// LS Electric XG5000 project: MODBUS_PR_3차프로젝트 최종최종
// PLC LSPLC
// module base 0 slot 0: 입출력 모듈:XBC-DR32H (DC 24V 입력, 릴레이 출력 32점)

PROGRAM 구동부_사본 (task: 스캔 프로그램)

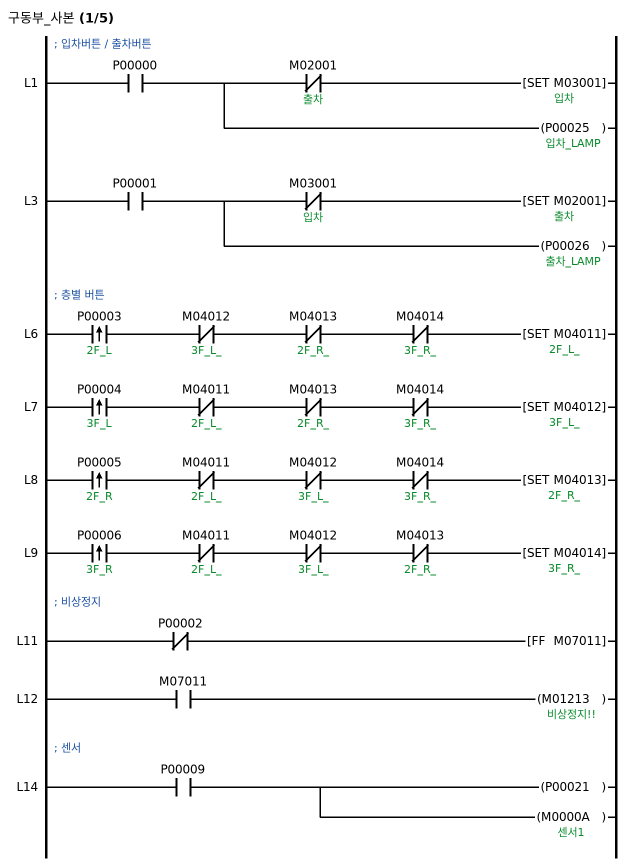
// 입차버튼 / 출차버튼
; L1
LOAD      P00000
MPUSH
AND NOT   M02001	// 출차
SET       M03001	// 입차
MPOP
OUT       P00025	// 입차_LAMP
; L3
LOAD      P00001
MPUSH
AND NOT   M03001	// 입차
SET       M02001	// 출차
MPOP
OUT       P00026	// 출차_LAMP
// 층별 버튼
; L6
LOADP     P00003	// 2F_L
AND NOT   M04012	// 3F_L_
AND NOT   M04013	// 2F_R_
AND NOT   M04014	// 3F_R_
SET       M04011	// 2F_L_
; L7
LOADP     P00004	// 3F_L
AND NOT   M04011	// 2F_L_
AND NOT   M04013	// 2F_R_
AND NOT   M04014	// 3F_R_
SET       M04012	// 3F_L_
; L8
LOADP     P00005	// 2F_R
AND NOT   M04011	// 2F_L_
AND NOT   M04012	// 3F_L_
AND NOT   M04014	// 3F_R_
SET       M04013	// 2F_R_
; L9
LOADP     P00006	// 3F_R
AND NOT   M04011	// 2F_L_
AND NOT   M04012	// 3F_L_
AND NOT   M04013	// 2F_R_
SET       M04014	// 3F_R_
// 비상정지
; L11
LOAD NOT  P00002
FF        M07011
; L12
LOAD      M07011
OUT       M01213	// 비상정지!!
// 센서
; L14
LOAD      P00009
OUT       P00021
OUT       M0000A	// 센서1

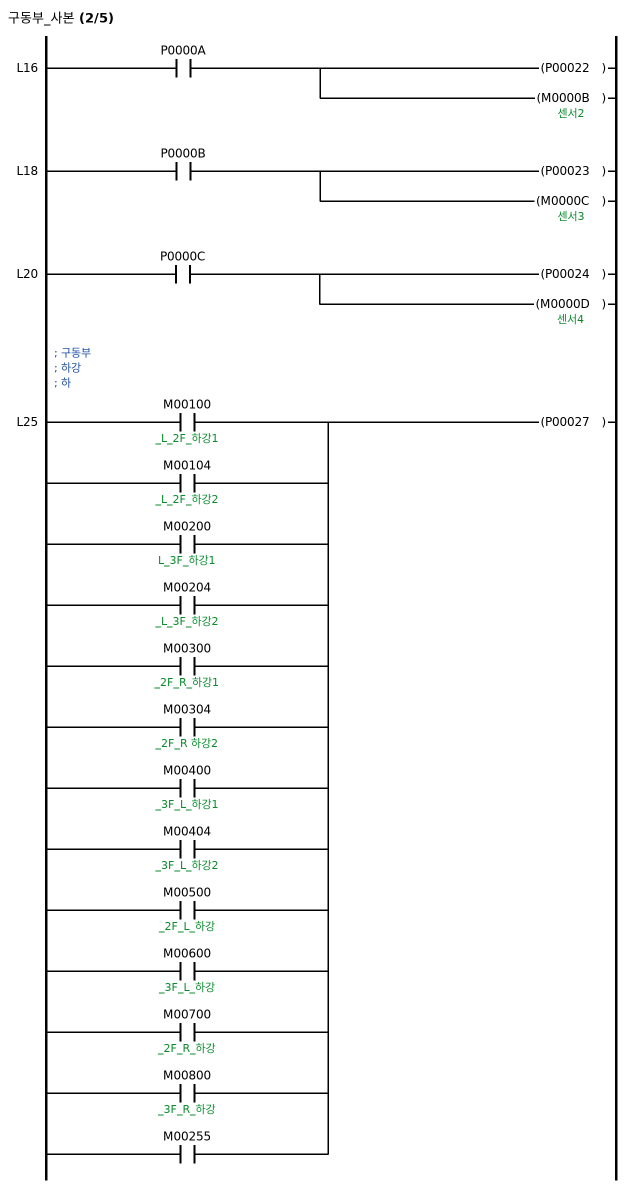
; L16
LOAD      P0000A
OUT       P00022
OUT       M0000B	// 센서2
; L18
LOAD      P0000B
OUT       P00023
OUT       M0000C	// 센서3
; L20
LOAD      P0000C
OUT       P00024
OUT       M0000D	// 센서4
// 구동부
// 하강
; L25
LOAD      M00100	// _L_2F_하강1
OR        M00104	// _L_2F_하강2
OR        M00200	// L_3F_하강1
OR        M00204	// _L_3F_하강2
OR        M00300	// _2F_R_하강1
OR        M00304	// _2F_R 하강2
OR        M00400	// _3F_L_하강1
OR        M00404	// _3F_L_하강2
OR        M00500	// _2F_L_하강
OR        M00600	// _3F_L_하강
OR        M00700	// _2F_R_하강
OR        M00800	// _3F_R_하강
OR        M00255
OUT       P00027
// output comment: 하

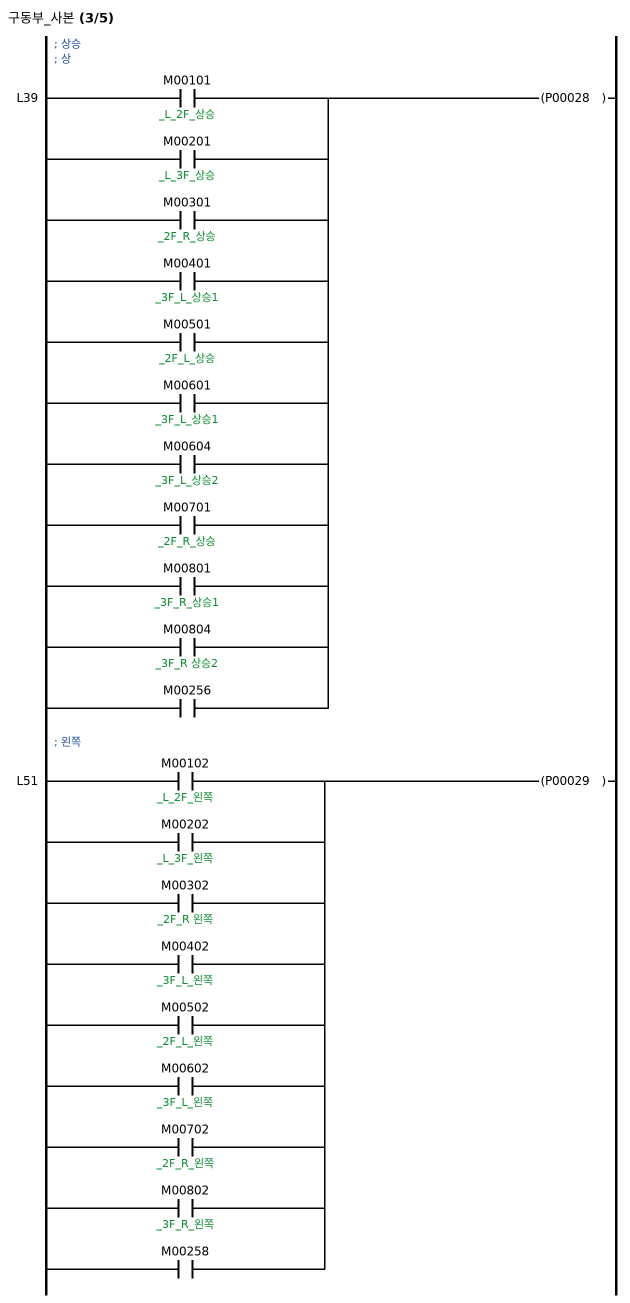
// 상승
; L39
LOAD      M00101	// _L_2F_상승
OR        M00201	// _L_3F_상승
OR        M00301	// _2F_R_상승
OR        M00401	// _3F_L_상승1
OR        M00501	// _2F_L_상승
OR        M00601	// _3F_L_상승1
OR        M00604	// _3F_L_상승2
OR        M00701	// _2F_R_상승
OR        M00801	// _3F_R_상승1
OR        M00804	// _3F_R 상승2
OR        M00256
OUT       P00028
// output comment: 상
// 왼쪽
; L51
LOAD      M00102	// _L_2F_왼쪽
OR        M00202	// _L_3F_왼쪽
OR        M00302	// _2F_R 왼쪽
OR        M00402	// _3F_L_왼쪽
OR        M00502	// _2F_L_왼쪽
OR        M00602	// _3F_L_왼쪽
OR        M00702	// _2F_R_왼쪽
OR        M00802	// _3F_R_왼쪽
OR        M00258
OUT       P00029

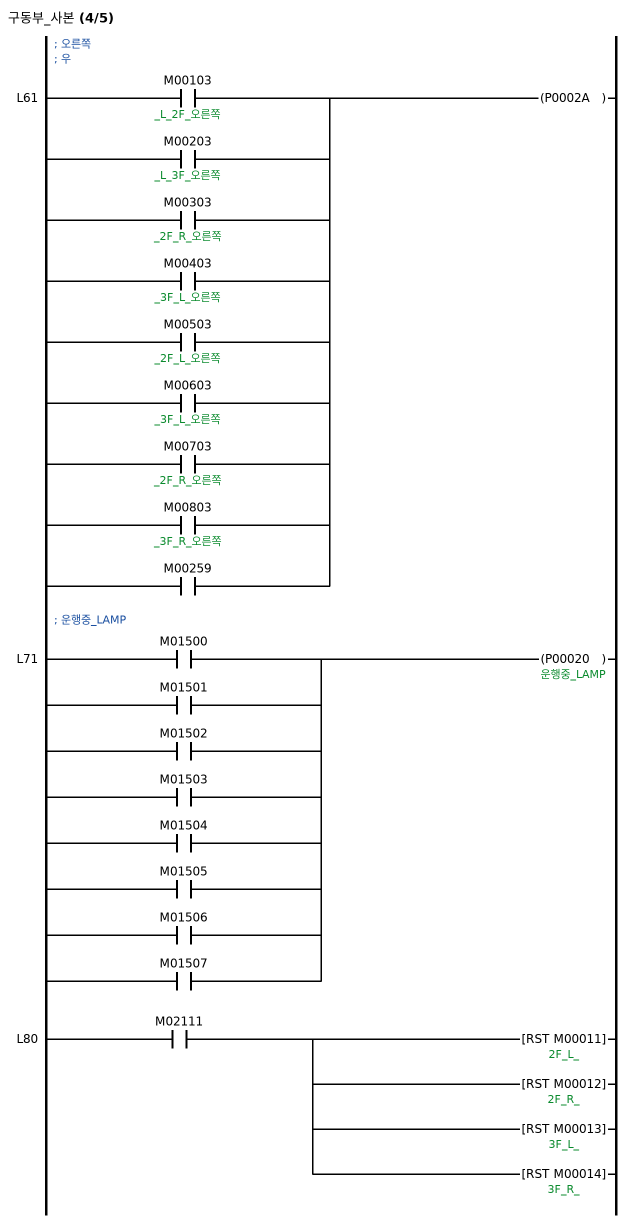
// 오른쪽
; L61
LOAD      M00103	// _L_2F_오른쪽
OR        M00203	// _L_3F_오른쪽
OR        M00303	// _2F_R_오른쪽
OR        M00403	// _3F_L_오른쪽
OR        M00503	// _2F_L_오른쪽
OR        M00603	// _3F_L_오른쪽
OR        M00703	// _2F_R_오른쪽
OR        M00803	// _3F_R_오른쪽
OR        M00259
OUT       P0002A
// output comment: 우
// 운행중_LAMP
; L71
LOAD      M01500
OR        M01501
OR        M01502
OR        M01503
OR        M01504
OR        M01505
OR        M01506
OR        M01507
OUT       P00020	// 운행중_LAMP
; L80
LOAD      M02111
RST       M00011	// 2F_L_
RST       M00012	// 2F_R_
RST       M00013	// 3F_L_
RST       M00014	// 3F_R_

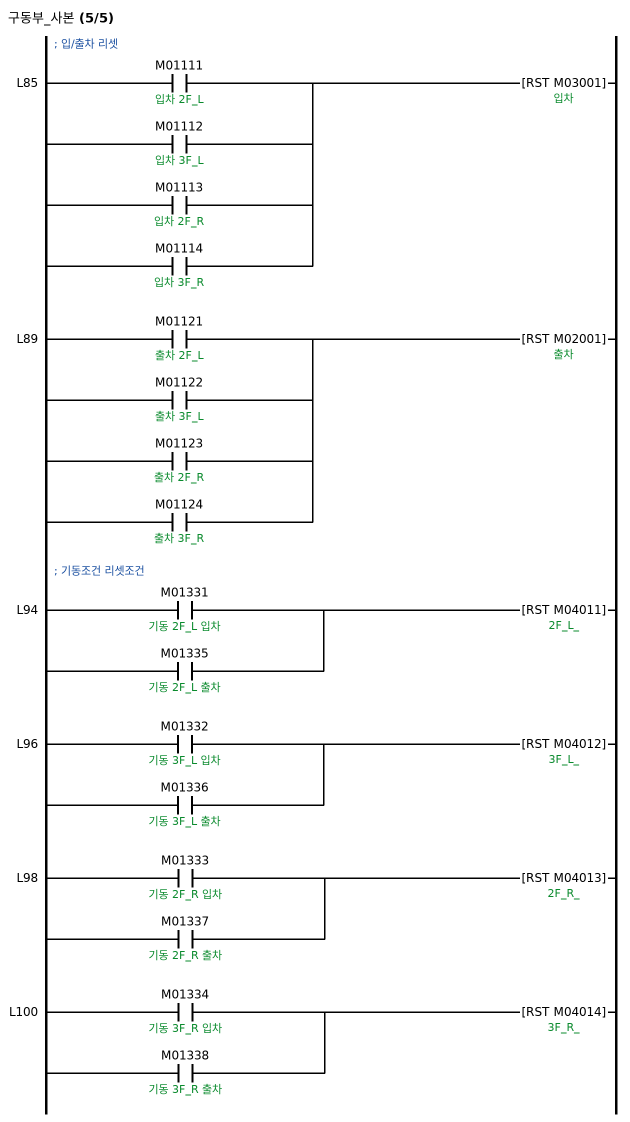
// 입/출차 리셋
; L85
LOAD      M01111	// 입차 2F_L 
OR        M01112	// 입차 3F_L
OR        M01113	// 입차 2F_R
OR        M01114	// 입차 3F_R
RST       M03001	// 입차
; L89
LOAD      M01121	// 출차 2F_L
OR        M01122	// 출차 3F_L
OR        M01123	// 출차 2F_R
OR        M01124	// 출차 3F_R
RST       M02001	// 출차
// 기동조건 리셋조건
; L94
LOAD      M01331	// 기동 2F_L 입차
OR        M01335	// 기동 2F_L 출차
RST       M04011	// 2F_L_
; L96
LOAD      M01332	// 기동 3F_L 입차
OR        M01336	// 기동 3F_L 출차
RST       M04012	// 3F_L_
; L98
LOAD      M01333	// 기동 2F_R 입차
OR        M01337	// 기동 2F_R 출차
RST       M04013	// 2F_R_
; L100
LOAD      M01334	// 기동 3F_R 입차
OR        M01338	// 기동 3F_R 출차
RST       M04014	// 3F_R_

PROGRAM 출차 (task: 스캔 프로그램)

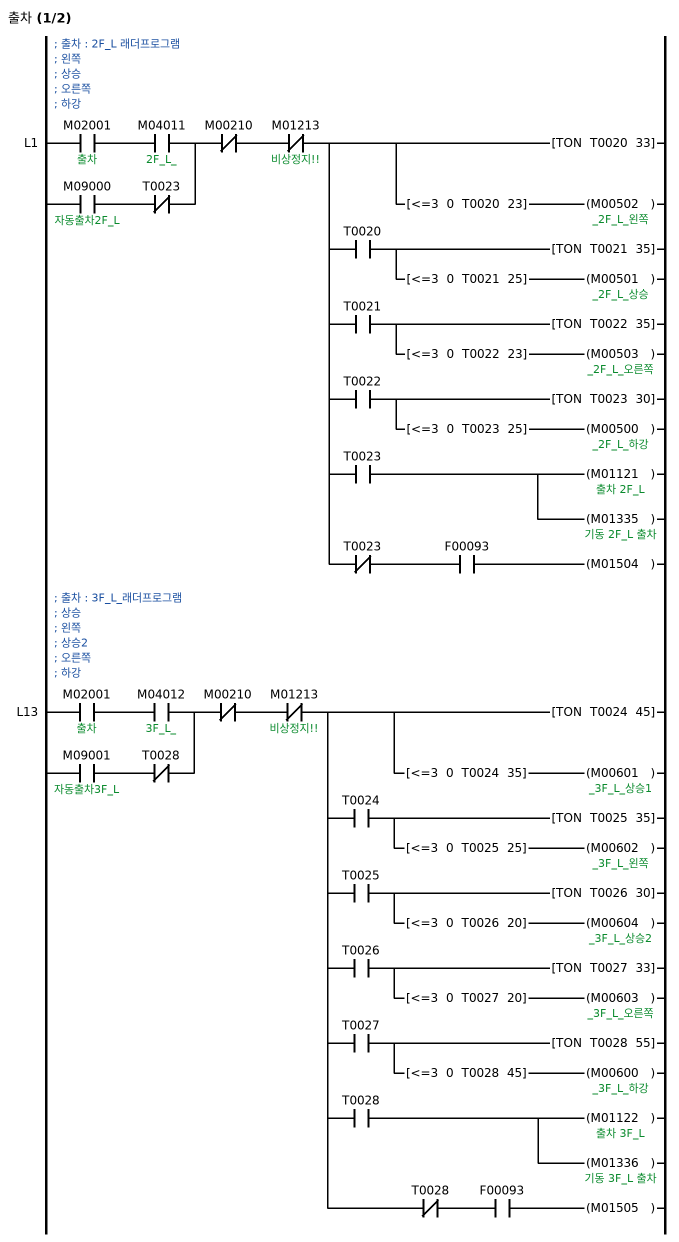
// 출차 : 2F_L 래더프로그램
; L1
LOAD      M02001	// 출차
AND       M04011	// 2F_L_
LOAD      M09000	// 자동출차2F_L
AND NOT   T0023
OR LOAD
AND NOT   M00210
AND NOT   M01213	// 비상정지!!
TON       T0020 33
MPUSH
AND<=3    0 T0020 23
OUT       M00502	// _2F_L_왼쪽
MLOAD
AND       T0020
TON       T0021 35
AND<=3    0 T0021 25
OUT       M00501	// _2F_L_상승
MLOAD
AND       T0021
TON       T0022 35
AND<=3    0 T0022 23
OUT       M00503	// _2F_L_오른쪽
MLOAD
AND       T0022
TON       T0023 30
AND<=3    0 T0023 25
OUT       M00500	// _2F_L_하강
MLOAD
AND       T0023
OUT       M01121	// 출차 2F_L
OUT       M01335	// 기동 2F_L 출차
MPOP
AND NOT   T0023
AND       F00093
OUT       M01504
// output comment: 왼쪽
// output comment: 상승
// output comment: 오른쪽
// output comment: 하강
// 출차 : 3F_L_래더프로그램
; L13
LOAD      M02001	// 출차
AND       M04012	// 3F_L_
LOAD      M09001	// 자동출차3F_L
AND NOT   T0028
OR LOAD
AND NOT   M00210
AND NOT   M01213	// 비상정지!!
TON       T0024 45
MPUSH
AND<=3    0 T0024 35
OUT       M00601	// _3F_L_상승1
MLOAD
AND       T0024
TON       T0025 35
AND<=3    0 T0025 25
OUT       M00602	// _3F_L_왼쪽
MLOAD
AND       T0025
TON       T0026 30
AND<=3    0 T0026 20
OUT       M00604	// _3F_L_상승2
MLOAD
AND       T0026
TON       T0027 33
AND<=3    0 T0027 20
OUT       M00603	// _3F_L_오른쪽
MLOAD
AND       T0027
TON       T0028 55
AND<=3    0 T0028 45
OUT       M00600	// _3F_L_하강
MLOAD
AND       T0028
OUT       M01122	// 출차 3F_L
OUT       M01336	// 기동 3F_L 출차
MPOP
AND NOT   T0028
AND       F00093
OUT       M01505
// output comment: 상승
// output comment: 왼쪽
// output comment: 상승2
// output comment: 오른쪽
// output comment: 하강

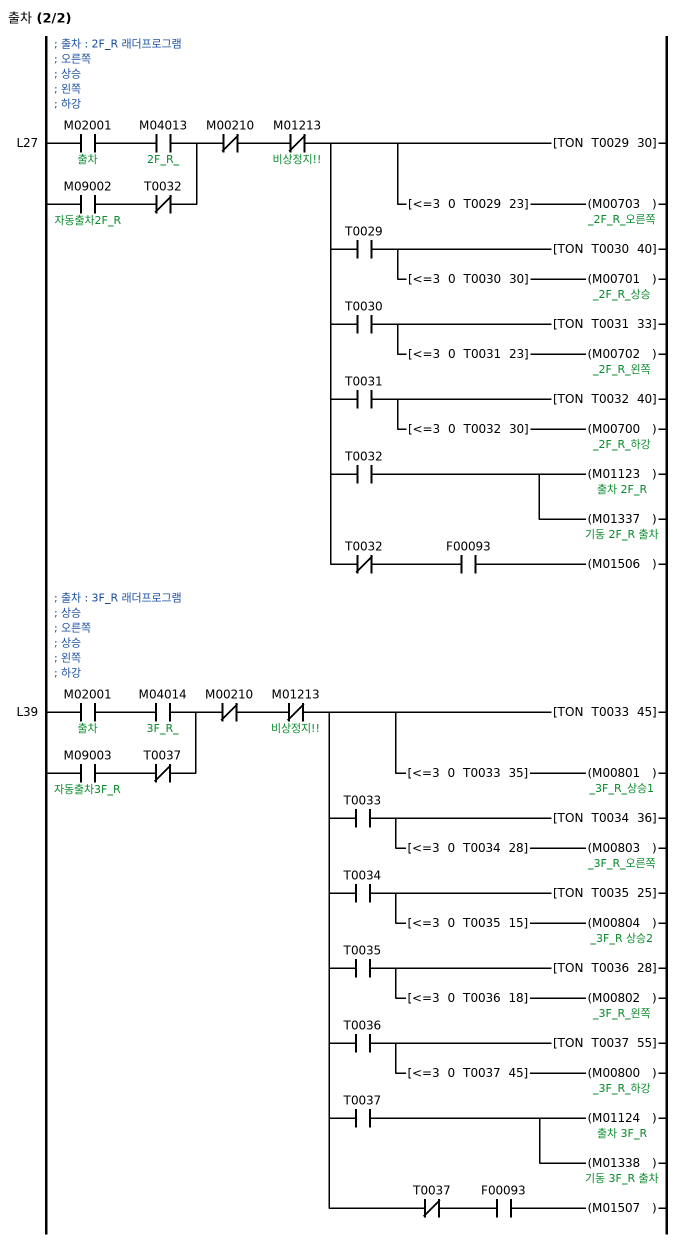
// 출차 : 2F_R 래더프로그램
; L27
LOAD      M02001	// 출차
AND       M04013	// 2F_R_
LOAD      M09002	// 자동출차2F_R
AND NOT   T0032
OR LOAD
AND NOT   M00210
AND NOT   M01213	// 비상정지!!
TON       T0029 30
MPUSH
AND<=3    0 T0029 23
OUT       M00703	// _2F_R_오른쪽
MLOAD
AND       T0029
TON       T0030 40
AND<=3    0 T0030 30
OUT       M00701	// _2F_R_상승
MLOAD
AND       T0030
TON       T0031 33
AND<=3    0 T0031 23
OUT       M00702	// _2F_R_왼쪽
MLOAD
AND       T0031
TON       T0032 40
AND<=3    0 T0032 30
OUT       M00700	// _2F_R_하강
MLOAD
AND       T0032
OUT       M01123	// 출차 2F_R
OUT       M01337	// 기동 2F_R 출차
MPOP
AND NOT   T0032
AND       F00093
OUT       M01506
// output comment: 오른쪽
// output comment: 상승
// output comment: 왼쪽
// output comment: 하강
// 출차 : 3F_R 래더프로그램
; L39
LOAD      M02001	// 출차
AND       M04014	// 3F_R_
LOAD      M09003	// 자동출차3F_R
AND NOT   T0037
OR LOAD
AND NOT   M00210
AND NOT   M01213	// 비상정지!!
TON       T0033 45
MPUSH
AND<=3    0 T0033 35
OUT       M00801	// _3F_R_상승1
MLOAD
AND       T0033
TON       T0034 36
AND<=3    0 T0034 28
OUT       M00803	// _3F_R_오른쪽
MLOAD
AND       T0034
TON       T0035 25
AND<=3    0 T0035 15
OUT       M00804	// _3F_R 상승2
MLOAD
AND       T0035
TON       T0036 28
AND<=3    0 T0036 18
OUT       M00802	// _3F_R_왼쪽
MLOAD
AND       T0036
TON       T0037 55
AND<=3    0 T0037 45
OUT       M00800	// _3F_R_하강
MLOAD
AND       T0037
OUT       M01124	// 출차 3F_R
OUT       M01338	// 기동 3F_R 출차
MPOP
AND NOT   T0037
AND       F00093
OUT       M01507
// output comment: 상승
// output comment: 오른쪽
// output comment: 상승
// output comment: 왼쪽
// output comment: 하강

PROGRAM 입차 (task: 스캔 프로그램)

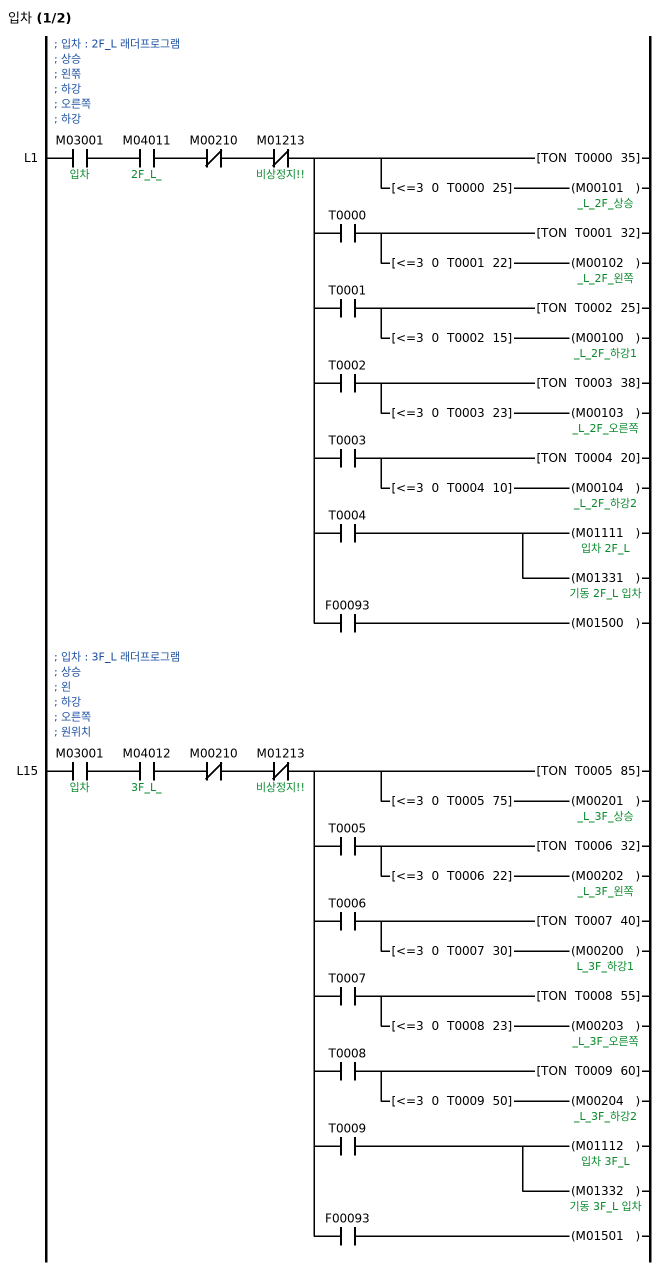
// 입차 : 2F_L 래더프로그램
; L1
LOAD      M03001	// 입차
AND       M04011	// 2F_L_
AND NOT   M00210
AND NOT   M01213	// 비상정지!!
TON       T0000 35
MPUSH
AND<=3    0 T0000 25
OUT       M00101	// _L_2F_상승
MLOAD
AND       T0000
TON       T0001 32
AND<=3    0 T0001 22
OUT       M00102	// _L_2F_왼쪽
MLOAD
AND       T0001
TON       T0002 25
AND<=3    0 T0002 15
OUT       M00100	// _L_2F_하강1
MLOAD
AND       T0002
TON       T0003 38
AND<=3    0 T0003 23
OUT       M00103	// _L_2F_오른쪽
MLOAD
AND       T0003
TON       T0004 20
AND<=3    0 T0004 10
OUT       M00104	// _L_2F_하강2
MLOAD
AND       T0004
OUT       M01111	// 입차 2F_L 
OUT       M01331	// 기동 2F_L 입차
MPOP
AND       F00093
OUT       M01500
// output comment: 상승
// output comment: 왼쪾
// output comment: 하강
// output comment: 오른쪽
// output comment: 하강
// 입차 : 3F_L 래더프로그램
; L15
LOAD      M03001	// 입차
AND       M04012	// 3F_L_
AND NOT   M00210
AND NOT   M01213	// 비상정지!!
TON       T0005 85
MPUSH
AND<=3    0 T0005 75
OUT       M00201	// _L_3F_상승
MLOAD
AND       T0005
TON       T0006 32
AND<=3    0 T0006 22
OUT       M00202	// _L_3F_왼쪽
MLOAD
AND       T0006
TON       T0007 40
AND<=3    0 T0007 30
OUT       M00200	// L_3F_하강1
MLOAD
AND       T0007
TON       T0008 55
AND<=3    0 T0008 23
OUT       M00203	// _L_3F_오른쪽
MLOAD
AND       T0008
TON       T0009 60
AND<=3    0 T0009 50
OUT       M00204	// _L_3F_하강2
MLOAD
AND       T0009
OUT       M01112	// 입차 3F_L
OUT       M01332	// 기동 3F_L 입차
MPOP
AND       F00093
OUT       M01501
// output comment: 상승
// output comment: 왼
// output comment: 하강
// output comment: 오른쪽
// output comment: 원위치

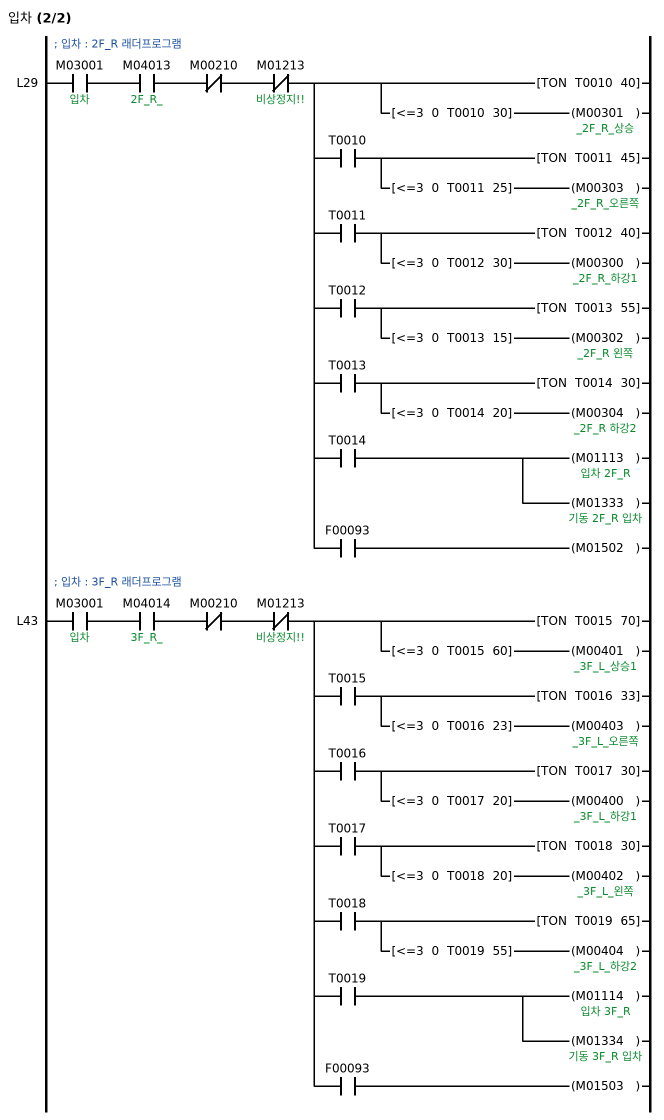
// 입차 : 2F_R 래더프로그램
; L29
LOAD      M03001	// 입차
AND       M04013	// 2F_R_
AND NOT   M00210
AND NOT   M01213	// 비상정지!!
TON       T0010 40
MPUSH
AND<=3    0 T0010 30
OUT       M00301	// _2F_R_상승
MLOAD
AND       T0010
TON       T0011 45
AND<=3    0 T0011 25
OUT       M00303	// _2F_R_오른쪽
MLOAD
AND       T0011
TON       T0012 40
AND<=3    0 T0012 30
OUT       M00300	// _2F_R_하강1
MLOAD
AND       T0012
TON       T0013 55
AND<=3    0 T0013 15
OUT       M00302	// _2F_R 왼쪽
MLOAD
AND       T0013
TON       T0014 30
AND<=3    0 T0014 20
OUT       M00304	// _2F_R 하강2
MLOAD
AND       T0014
OUT       M01113	// 입차 2F_R
OUT       M01333	// 기동 2F_R 입차
MPOP
AND       F00093
OUT       M01502
// 입차 : 3F_R 래더프로그램
; L43
LOAD      M03001	// 입차
AND       M04014	// 3F_R_
AND NOT   M00210
AND NOT   M01213	// 비상정지!!
TON       T0015 70
MPUSH
AND<=3    0 T0015 60
OUT       M00401	// _3F_L_상승1
MLOAD
AND       T0015
TON       T0016 33
AND<=3    0 T0016 23
OUT       M00403	// _3F_L_오른쪽
MLOAD
AND       T0016
TON       T0017 30
AND<=3    0 T0017 20
OUT       M00400	// _3F_L_하강1
MLOAD
AND       T0017
TON       T0018 30
AND<=3    0 T0018 20
OUT       M00402	// _3F_L_왼쪽
MLOAD
AND       T0018
TON       T0019 65
AND<=3    0 T0019 55
OUT       M00404	// _3F_L_하강2
MLOAD
AND       T0019
OUT       M01114	// 입차 3F_R
OUT       M01334	// 기동 3F_R 입차
MPOP
AND       F00093
OUT       M01503

PROGRAM 00.Initialize (task: 스캔 프로그램)

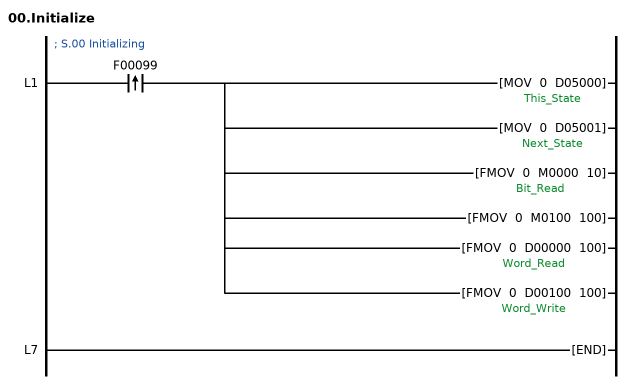
// S.00 Initializing
; L1
LOADP     F00099
MOV       0 D05000	// This_State
MOV       0 D05001	// Next_State
FMOV      0 M0000 10	// Bit_Read
FMOV      0 M0100 100
FMOV      0 D00000 100	// Word_Read
FMOV      0 D00100 100	// Word_Write
; L7
END

PROGRAM 10.Main (task: 스캔 프로그램)

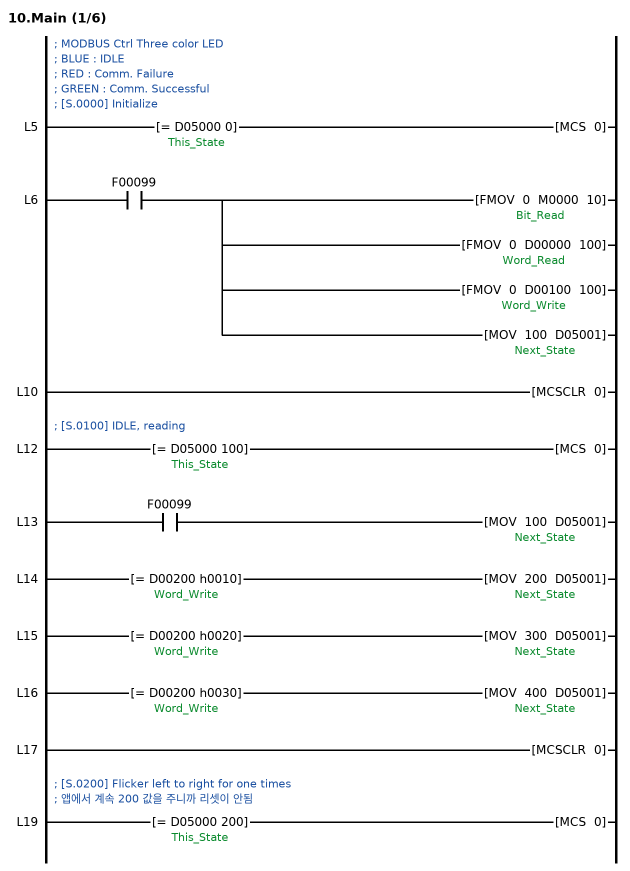
// MODBUS Ctrl Three color LED
// BLUE : IDLE
// RED : Comm. Failure
// GREEN : Comm. Successful
// [S.0000] Initialize
; L5
LOAD=     D05000 0	// This_State
MCS       0
; L6
LOAD      F00099
FMOV      0 M0000 10	// Bit_Read
FMOV      0 D00000 100	// Word_Read
FMOV      0 D00100 100	// Word_Write
MOV       100 D05001	// Next_State
; L10
MCSCLR    0
// [S.0100] IDLE, reading
; L12
LOAD=     D05000 100	// This_State
MCS       0
; L13
LOAD      F00099
MOV       100 D05001	// Next_State
; L14
LOAD=     D00200 h0010	// Word_Write
MOV       200 D05001	// Next_State
; L15
LOAD=     D00200 h0020	// Word_Write
MOV       300 D05001	// Next_State
; L16
LOAD=     D00200 h0030	// Word_Write
MOV       400 D05001	// Next_State
; L17
MCSCLR    0
// [S.0200] Flicker left to right for one times
; L19
LOAD=     D05000 200	// This_State
MCS       0
// output comment: 앱에서 계속 200 값을 주니까 리셋이 안됨

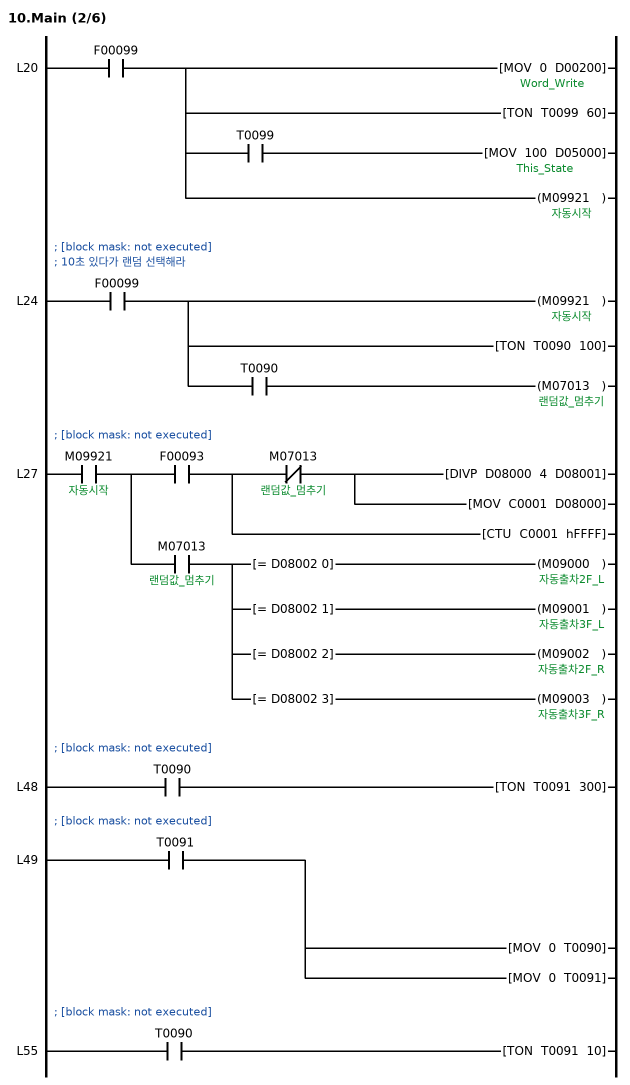
; L20
LOAD      F00099
MOV       0 D00200	// Word_Write
TON       T0099 60
MPUSH
AND       T0099
MOV       100 D05000	// This_State
MPOP
OUT       M09921	// 자동시작
; L24 (block mask: not executed)
LOAD      F00099
OUT       M09921	// 자동시작
TON       T0090 100
AND       T0090
OUT       M07013	// 랜덤값_멈추기
// output comment: 10초 있다가 랜덤 선택해라
; L27 (block mask: not executed)
LOAD      M09921	// 자동시작
MPUSH
AND       F00093
MPUSH
AND NOT   M07013	// 랜덤값_멈추기
DIVP      D08000 4 D08001
MOV       C0001 D08000
MPOP
CTU       C0001 hFFFF
MPOP
AND       M07013	// 랜덤값_멈추기
MPUSH
AND=      D08002 0
OUT       M09000	// 자동출차2F_L
MLOAD
AND=      D08002 1
OUT       M09001	// 자동출차3F_L
MLOAD
AND=      D08002 2
OUT       M09002	// 자동출차2F_R
MPOP
AND=      D08002 3
OUT       M09003	// 자동출차3F_R
; L48 (block mask: not executed)
LOAD      T0090
TON       T0091 300
; L49 (block mask: not executed)
LOAD      T0091
MOV       0 T0090
MOV       0 T0091
; L55 (block mask: not executed)
LOAD      T0090
TON       T0091 10

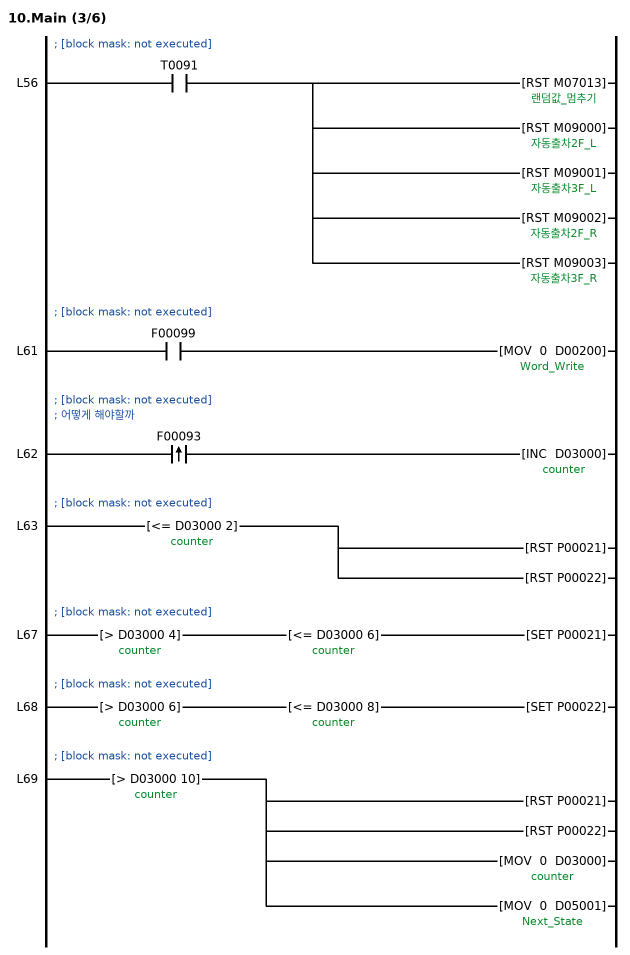
; L56 (block mask: not executed)
LOAD      T0091
RST       M07013	// 랜덤값_멈추기
RST       M09000	// 자동출차2F_L
RST       M09001	// 자동출차3F_L
RST       M09002	// 자동출차2F_R
RST       M09003	// 자동출차3F_R
; L61 (block mask: not executed)
LOAD      F00099
MOV       0 D00200	// Word_Write
; L62 (block mask: not executed)
LOADP     F00093
INC       D03000	// counter
// output comment: 어떻게 해야할까
; L63 (block mask: not executed)
LOAD<=    D03000 2	// counter
RST       P00021
RST       P00022
; L67 (block mask: not executed)
LOAD>     D03000 4	// counter
AND<=     D03000 6	// counter
SET       P00021
; L68 (block mask: not executed)
LOAD>     D03000 6	// counter
AND<=     D03000 8	// counter
SET       P00022
; L69 (block mask: not executed)
LOAD>     D03000 10	// counter
RST       P00021
RST       P00022
MOV       0 D03000	// counter
MOV       0 D05001	// Next_State

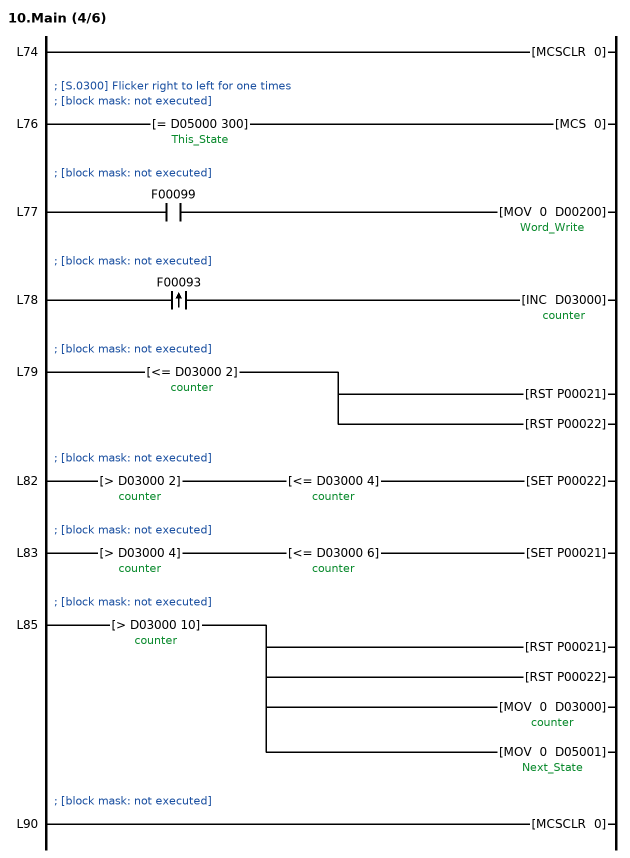
; L74
MCSCLR    0
// [S.0300] Flicker right to left for one times
; L76 (block mask: not executed)
LOAD=     D05000 300	// This_State
MCS       0
; L77 (block mask: not executed)
LOAD      F00099
MOV       0 D00200	// Word_Write
; L78 (block mask: not executed)
LOADP     F00093
INC       D03000	// counter
; L79 (block mask: not executed)
LOAD<=    D03000 2	// counter
RST       P00021
RST       P00022
; L82 (block mask: not executed)
LOAD>     D03000 2	// counter
AND<=     D03000 4	// counter
SET       P00022
; L83 (block mask: not executed)
LOAD>     D03000 4	// counter
AND<=     D03000 6	// counter
SET       P00021
; L85 (block mask: not executed)
LOAD>     D03000 10	// counter
RST       P00021
RST       P00022
MOV       0 D03000	// counter
MOV       0 D05001	// Next_State
; L90 (block mask: not executed)
MCSCLR    0

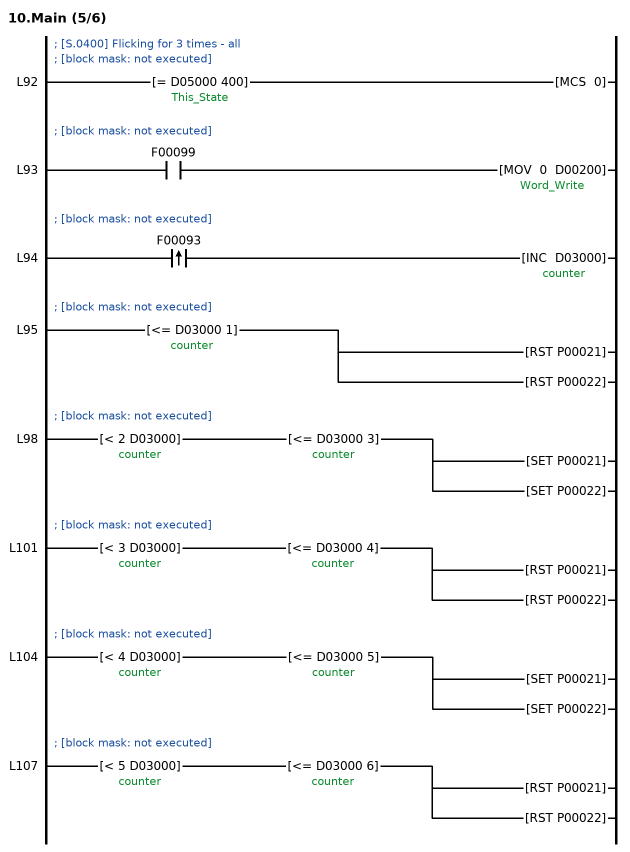
// [S.0400] Flicking for 3 times - all
; L92 (block mask: not executed)
LOAD=     D05000 400	// This_State
MCS       0
; L93 (block mask: not executed)
LOAD      F00099
MOV       0 D00200	// Word_Write
; L94 (block mask: not executed)
LOADP     F00093
INC       D03000	// counter
; L95 (block mask: not executed)
LOAD<=    D03000 1	// counter
RST       P00021
RST       P00022
; L98 (block mask: not executed)
LOAD<     2 D03000	// counter
AND<=     D03000 3	// counter
SET       P00021
SET       P00022
; L101 (block mask: not executed)
LOAD<     3 D03000	// counter
AND<=     D03000 4	// counter
RST       P00021
RST       P00022
; L104 (block mask: not executed)
LOAD<     4 D03000	// counter
AND<=     D03000 5	// counter
SET       P00021
SET       P00022
; L107 (block mask: not executed)
LOAD<     5 D03000	// counter
AND<=     D03000 6	// counter
RST       P00021
RST       P00022

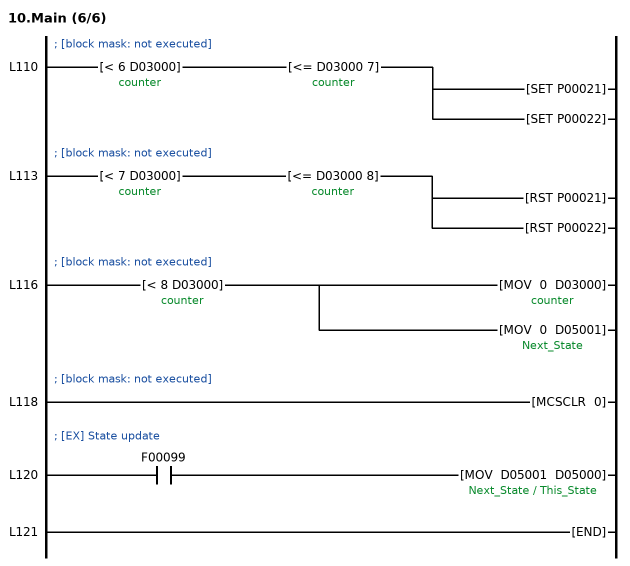
; L110 (block mask: not executed)
LOAD<     6 D03000	// counter
AND<=     D03000 7	// counter
SET       P00021
SET       P00022
; L113 (block mask: not executed)
LOAD<     7 D03000	// counter
AND<=     D03000 8	// counter
RST       P00021
RST       P00022
; L116 (block mask: not executed)
LOAD<     8 D03000	// counter
MOV       0 D03000	// counter
MOV       0 D05001	// Next_State
; L118 (block mask: not executed)
MCSCLR    0
// [EX] State update
; L120
LOAD      F00099
MOV       D05001 D05000	// Next_State / This_State
; L121
END

PROGRAM 20.IO_Ctrl (task: 스캔 프로그램)

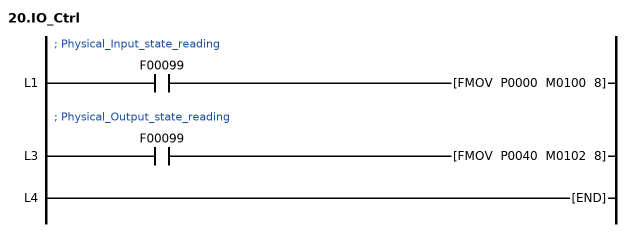
// Physical_Input_state_reading
; L1
LOAD      F00099
FMOV      P0000 M0100 8
// Physical_Output_state_reading
; L3
LOAD      F00099
FMOV      P0040 M0102 8
; L4
END

PROGRAM random_random (task: 스캔 프로그램)

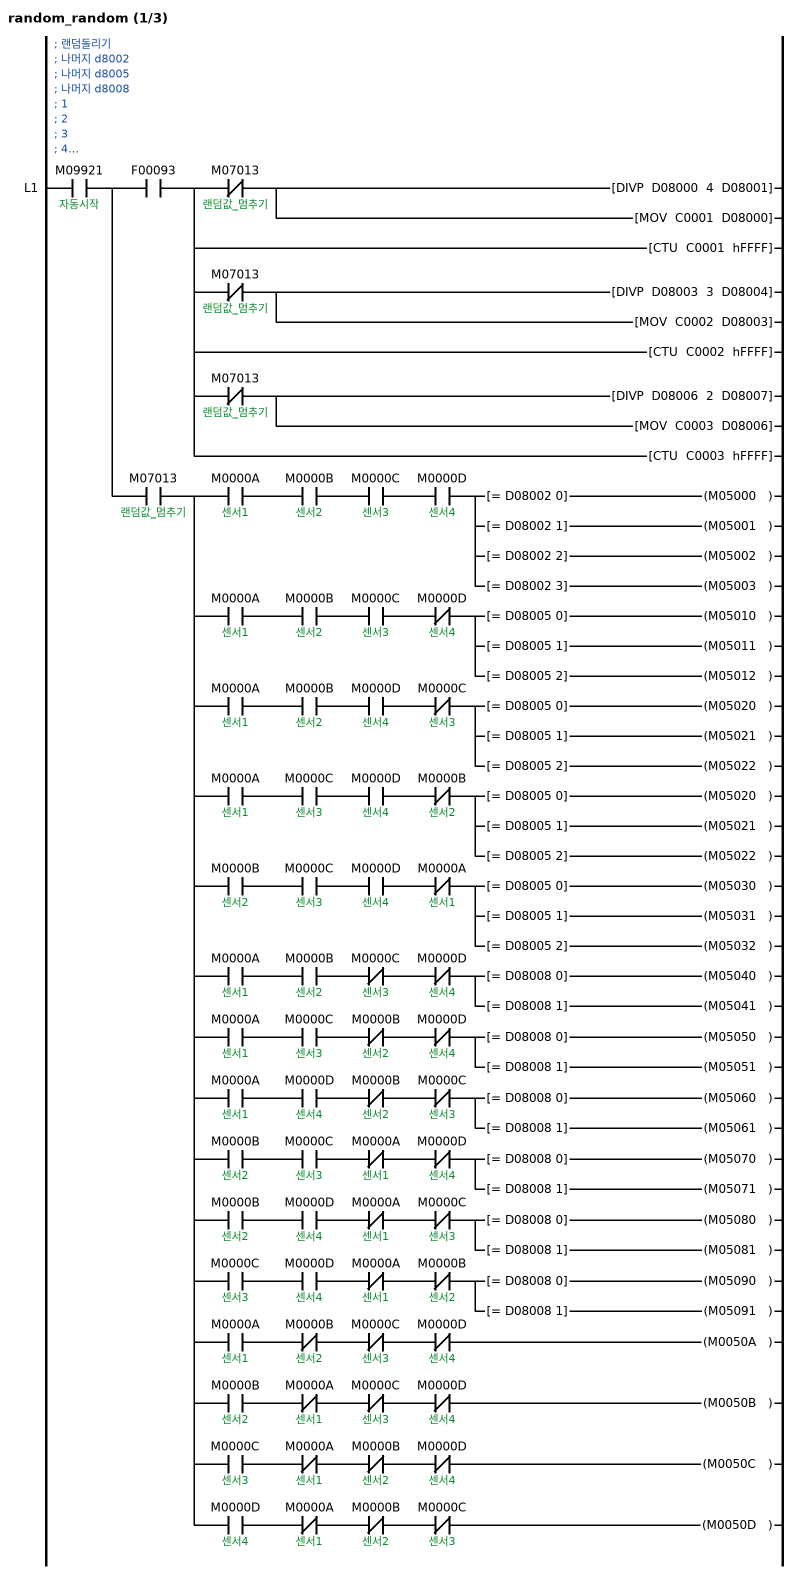
// 랜덤돌리기
; L1
LOAD      M09921	// 자동시작
MPUSH
AND       F00093
MPUSH
AND NOT   M07013	// 랜덤값_멈추기
DIVP      D08000 4 D08001
MOV       C0001 D08000
MLOAD
CTU       C0001 hFFFF
AND NOT   M07013	// 랜덤값_멈추기
DIVP      D08003 3 D08004
MOV       C0002 D08003
MLOAD
CTU       C0002 hFFFF
AND NOT   M07013	// 랜덤값_멈추기
DIVP      D08006 2 D08007
MOV       C0003 D08006
MPOP
CTU       C0003 hFFFF
MPOP
AND       M07013	// 랜덤값_멈추기
MPUSH
AND       M0000A	// 센서1
AND       M0000B	// 센서2
AND       M0000C	// 센서3
AND       M0000D	// 센서4
MPUSH
AND=      D08002 0
OUT       M05000
MLOAD
AND=      D08002 1
OUT       M05001
MLOAD
AND=      D08002 2
OUT       M05002
MPOP
AND=      D08002 3
OUT       M05003
MLOAD
AND       M0000A	// 센서1
AND       M0000B	// 센서2
AND       M0000C	// 센서3
AND NOT   M0000D	// 센서4
MPUSH
AND=      D08005 0
OUT       M05010
MLOAD
AND=      D08005 1
OUT       M05011
MPOP
AND=      D08005 2
OUT       M05012
MLOAD
AND       M0000A	// 센서1
AND       M0000B	// 센서2
AND       M0000D	// 센서4
AND NOT   M0000C	// 센서3
MPUSH
AND=      D08005 0
OUT       M05020
MLOAD
AND=      D08005 1
OUT       M05021
MPOP
AND=      D08005 2
OUT       M05022
MLOAD
AND       M0000A	// 센서1
AND       M0000C	// 센서3
AND       M0000D	// 센서4
AND NOT   M0000B	// 센서2
MPUSH
AND=      D08005 0
OUT       M05020
MLOAD
AND=      D08005 1
OUT       M05021
MPOP
AND=      D08005 2
OUT       M05022
MLOAD
AND       M0000B	// 센서2
AND       M0000C	// 센서3
AND       M0000D	// 센서4
AND NOT   M0000A	// 센서1
MPUSH
AND=      D08005 0
OUT       M05030
MLOAD
AND=      D08005 1
OUT       M05031
MPOP
AND=      D08005 2
OUT       M05032
MLOAD
AND       M0000A	// 센서1
AND       M0000B	// 센서2
AND NOT   M0000C	// 센서3
AND NOT   M0000D	// 센서4
MPUSH
AND=      D08008 0
OUT       M05040
MPOP
AND=      D08008 1
OUT       M05041
MLOAD
AND       M0000A	// 센서1
AND       M0000C	// 센서3
AND NOT   M0000B	// 센서2
AND NOT   M0000D	// 센서4
MPUSH
AND=      D08008 0
OUT       M05050
MPOP
AND=      D08008 1
OUT       M05051
MLOAD
AND       M0000A	// 센서1
AND       M0000D	// 센서4
AND NOT   M0000B	// 센서2
AND NOT   M0000C	// 센서3
MPUSH
AND=      D08008 0
OUT       M05060
MPOP
AND=      D08008 1
OUT       M05061
MLOAD
AND       M0000B	// 센서2
AND       M0000C	// 센서3
AND NOT   M0000A	// 센서1
AND NOT   M0000D	// 센서4
MPUSH
AND=      D08008 0
OUT       M05070
MPOP
AND=      D08008 1
OUT       M05071
MLOAD
AND       M0000B	// 센서2
AND       M0000D	// 센서4
AND NOT   M0000A	// 센서1
AND NOT   M0000C	// 센서3
MPUSH
AND=      D08008 0
OUT       M05080
MPOP
AND=      D08008 1
OUT       M05081
MLOAD
AND       M0000C	// 센서3
AND       M0000D	// 센서4
AND NOT   M0000A	// 센서1
AND NOT   M0000B	// 센서2
MPUSH
AND=      D08008 0
OUT       M05090
MPOP
AND=      D08008 1
OUT       M05091
MLOAD
AND       M0000A	// 센서1
AND NOT   M0000B	// 센서2
AND NOT   M0000C	// 센서3
AND NOT   M0000D	// 센서4
OUT       M0050A
MLOAD
AND       M0000B	// 센서2
AND NOT   M0000A	// 센서1
AND NOT   M0000C	// 센서3
AND NOT   M0000D	// 센서4
OUT       M0050B
MLOAD
AND       M0000C	// 센서3
AND NOT   M0000A	// 센서1
AND NOT   M0000B	// 센서2
AND NOT   M0000D	// 센서4
OUT       M0050C
MPOP
AND       M0000D	// 센서4
AND NOT   M0000A	// 센서1
AND NOT   M0000B	// 센서2
AND NOT   M0000C	// 센서3
OUT       M0050D
// output comment: 나머지 d8002
// output comment: 나머지 d8005
// output comment: 나머지 d8008
// output comment: 1
// output comment: 2
// output comment: 3
// output comment: 4
// output comment: 1
// output comment: 2
// output comment: 3
// output comment: 1
// output comment: 2
// output comment: 4
// output comment: 1
// output comment: 3
// output comment: 4
// output comment: 2
// output comment: 3
// output comment: 4
// output comment: 1
// output comment: 2
// output comment: 1
// output comment: 3
// output comment: 1
// output comment: 4
// output comment: 2
// output comment: 3
// output comment: 2
// output comment: 4
// output comment: 3
// output comment: 4

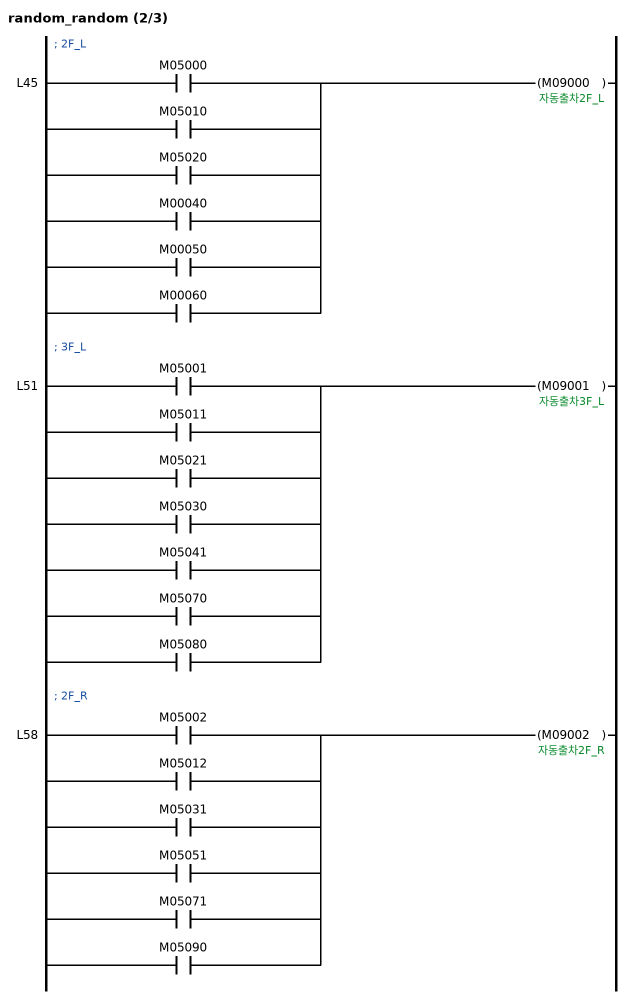
; L45
LOAD      M05000
OR        M05010
OR        M05020
OR        M00040
OR        M00050
OR        M00060
OUT       M09000	// 자동출차2F_L
// output comment: 2F_L
; L51
LOAD      M05001
OR        M05011
OR        M05021
OR        M05030
OR        M05041
OR        M05070
OR        M05080
OUT       M09001	// 자동출차3F_L
// output comment: 3F_L
; L58
LOAD      M05002
OR        M05012
OR        M05031
OR        M05051
OR        M05071
OR        M05090
OUT       M09002	// 자동출차2F_R
// output comment: 2F_R

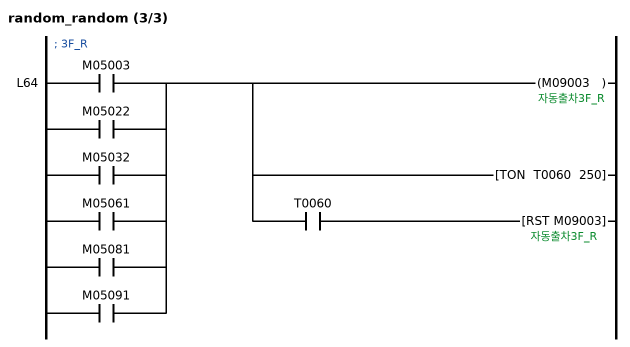
; L64
LOAD      M05003
OR        M05022
OR        M05032
OR        M05061
OR        M05081
OR        M05091
OUT       M09003	// 자동출차3F_R
TON       T0060 250
AND       T0060
RST       M09003	// 자동출차3F_R
// output comment: 3F_R

VARIABLES AND COMMENTS (devices not used above)
M00112	BIT	상승2
M01342	BIT	비상정지
M01351	BIT	비상정지
M01352	BIT	4개중에 하나 고르기
M01353	BIT	2F_L_py신호
M01354	BIT	3F_L_py신호
M01355	BIT	2F_R_py신호
M01356	BIT	3F_R_py신호
M01359	BIT	비상정지버튼
M0135A	BIT	2F_L_버튼
M0135B	BIT	2F_R_버튼
M0135C	BIT	3F_L_버튼
M0135D	BIT	3F_R_버튼
M0135E	BIT	센서 2F_L
M0135F	BIT	센서 3F_L
M01360	BIT	센서 2F_R
M01361	BIT	센서 3F_R
M01362	BIT	운행중_LAMP
M01363	BIT	LAMP_2F_L 
M01364	BIT	LAMP_3F_L
M01365	BIT	LAMP_2F_R
M01366	BIT	LAMP_3F_R 
M01367	BIT	하강
M01368	BIT	상승
M01369	BIT	왼쪽
M0136A	BIT	우측
M00902	BIT	_L_2F_왼쪽
M01011	BIT	 2F_L
M01012	BIT	 3F_L
M01013	BIT	 2F_R
M01014	BIT	차 3F_R
M01021	BIT	 2F_L 
M01022	BIT	 3F_L
M01023	BIT	 3F_R
M01024	BIT	 3F_R
M01343	BIT	 2F_L 운행중_LAMP
M01344	BIT	 3F_L 운행중_LAMP
M01345	BIT	 2F_R 운행중_LAMP
M01346	BIT	 3F_R 운행중_LAMP
M01347	BIT	 2F_L 운행중_LAMP
M01348	BIT	 3F_L 운행중_LAMP
M01349	BIT	 2F_R 운행중_LAMP
M0134A	BIT	 3F_R 운행중_LAMP
M0134D	BIT	2F_L 
M0134E	BIT	3F_L 
M0134F	BIT	2F_R 
M01350	BIT	3F_R 
M01357	BIT	버튼
M01358	BIT	버튼
M00091	BIT	\